// TwinCAT 3 PLC project Application
// ProgramVersion: 3.1.4022.2
// libraries:
//   Tc2_MC2, * (Beckhoff Automation GmbH)
//   Tc2_Standard, * (Beckhoff Automation GmbH)
//   Tc2_System, * (Beckhoff Automation GmbH)
//   Tc3_HBI_MC2, * (BeckHoff)
//   Tc3_Module, * (Beckhoff Automation GmbH)
// project tree:
//   / PlcTask.TcTTO
//   POUs/ MAIN.TcPOU, ST_Axis.TcDUT
// real-time tasks:
//   TASK PlcTask: cycle T#10ms, priority 20, ADS port 350
// motion (NC):
//   TASK NC-Task 1 SAF: cycle T#2ms, priority 4, ADS port 501
//   TASK NC-Task 1 SVB: cycle T#10ms, priority 8, ADS port 511
//   AXIS Axis 1 (id 1)
//     OtherSettings: AllowMotionCmdToSlave=true
//     encoder EncType=1
//     drive DrvType=5
//       Analog: ScaleFactorActTorque=0.1
//     controller CtrType=1
//       CtrPara: PriorControlFactor=1
//         Observer: BandWidth=20
//   AXIS Axis 2 (id 2)
//     OtherSettings: AllowMotionCmdToSlave=true
//     encoder EncType=1
//     drive DrvType=5
//       Analog: ScaleFactorActTorque=0.1
//     controller CtrType=1
//       CtrPara: PriorControlFactor=1
//         Observer: BandWidth=20
//   AXIS Axis 3 (id 3)
//     OtherSettings: AllowMotionCmdToSlave=true
//     encoder EncType=1
//     drive DrvType=5
//       Analog: ScaleFactorActTorque=0.1
//     controller CtrType=1
//       CtrPara: PriorControlFactor=1
//         Observer: BandWidth=20
// variable links:
//   Application/Application Instance <-> NC-Task 1 SAF/Axes/Axis 1
//     PlcTask Inputs/MAIN.fbAxis[0]._stAXIS_REF.NcToPlc <-> Outputs/ToPlc
//     PlcTask Outputs/MAIN.fbAxis[0]._stAXIS_REF.PlcToNc <-> Inputs/FromPlc
//   Application/Application Instance <-> NC-Task 1 SAF/Axes/Axis 2
//     PlcTask Inputs/MAIN.fbAxis[1]._stAXIS_REF.NcToPlc <-> Outputs/ToPlc
//     PlcTask Outputs/MAIN.fbAxis[1]._stAXIS_REF.PlcToNc <-> Inputs/FromPlc
//   Application/Application Instance <-> NC-Task 1 SAF/Axes/Axis 3
//     PlcTask Inputs/MAIN.fbAxis[2]._stAXIS_REF.NcToPlc <-> Outputs/ToPlc
//     PlcTask Outputs/MAIN.fbAxis[2]._stAXIS_REF.PlcToNc <-> Inputs/FromPlc

CONFIGURATION Application
    RESOURCE PLC ON TwinCAT3
        TASK PlcTask(INTERVAL := T#10ms, PRIORITY := 20);
        PROGRAM MAIN WITH PlcTask : MAIN;
    END_RESOURCE
END_CONFIGURATION

// ---- POUs/ST_Axis.TcDUT
TYPE ST_Axis :
STRUCT
	bEnable: BOOL;
	bEnable_Negative: BOOL;
	bEnable_Positive: BOOL;
	lrOverride: LREAL;
	bReset	: BOOL;
	bE_Stop: BOOL;
	bE_StopDelay: BOOL;
	bHome: BOOL;
	bCalibrationCam	: BOOL;
	lrHomePosition	: LREAL;
	bHalt	: BOOL;
	bStop	: BOOL;
	bAbsMove	: BOOL;
	lrAbsPosition	: LREAL;
	lrAbsVelocity	: LREAL;
	bRelMove	: BOOL;
	lrRelDistance	: LREAL;
	lrRelVelocity	: LREAL;
	bMoveVelo	: BOOL;
	lrVeloVelocity	: LREAL;
	bJogForward: BOOL;
	bJogBackwards: BOOL;
	lrJogVelocity	: LREAL;
	bSetDynamic		: BOOL;
	lrAcceleration	: LREAL;
	lrDecelaration	: LREAL;
	lrJerk			: LREAL;
	arr_nStatus	: ARRAY[1..10] OF UDINT;	

	//Vanessa added
	lrActPos : LREAL;
	lrActVelo : LREAL;
	bReady : BOOL;
	nVeloDirection : INT;
	nErrId : UDINT;
END_STRUCT
END_TYPE

// ---- POUs/MAIN.TcPOU
PROGRAM MAIN
VAR
	nAlive: INT;
	// Axis Instance
	fbAxis: ARRAY[0..2] OF Tc3_HBI_MC2.FB_MC2_Basic;
	
	bCalibrationCam : BOOL; //home sensor
	stAxis: ARRAY[0..2] OF ST_Axis;
	i: INT;
	
	//Input
	bInput1 : BOOL;
	bInput2 : BOOL;
	bInput3 : BOOL;
	bInput4 : BOOL;
	bInput5 : BOOL;
	bInput6 : BOOL;
	bInput7 : BOOL;
	bInput8 : BOOL;
	bInput9 : BOOL;
	bInput10 : BOOL;
	
	//Output
	bOutput1 : BOOL;
	bOutput2 : BOOL;
	bOutput3 : BOOL;
	bOutput4 : BOOL;
	bOutput5 : BOOL;
	bOutput6 : BOOL;
	bOutput7 : BOOL;
	bOutput8 : BOOL;
	bOutput9 : BOOL;
	bOutput10 : BOOL;
	
END_VAR

nAlive:= nAlive +1;

FOR i:= 0 TO 2 DO
	
//************************************
// Call methods
//************************************
stAxis[i].arr_nStatus[1]:= fbAxis[i].M_nMC_Power(bEnable:= stAxis[i].bEnable, bE_Stop:= stAxis[i].bE_Stop, 									// Enable
							bE_StopDelay:= stAxis[i].bE_StopDelay, bEnable_Positive:= stAxis[i].bEnable_Positive, 
							bEnable_Negative:= stAxis[i].bEnable_Negative);							
stAxis[i].arr_nStatus[2]:= fbAxis[i].M_nReset(bExecute:= stAxis[i].bReset);																// Reset
stAxis[i].arr_nStatus[3]:= fbAxis[i].M_nMC_Halt(bExecute:= stAxis[i].bHalt);																// Halt
stAxis[i].arr_nStatus[4]:= fbAxis[i].M_nMC_Stop(bExecute:= stAxis[i].bStop);																// Stop
stAxis[i].arr_nStatus[5]:= fbAxis[i].M_nMC_Home(bExecute:= stAxis[i].bHome, lrPosition:= stAxis[i].lrHomePosition, 							// Home
											bCalibrationCam:= stAxis[i].bCalibrationCam, eHomingMode:= MC_DefaultHoming);		
stAxis[i].arr_nStatus[6]:= fbAxis[i].M_nMC_MoveAbsolute(bExecute:= stAxis[i].bAbsMove, lrPosition:= stAxis[i].lrAbsPosition, 				// Absolute
													lrVelocity:= stAxis[i].lrAbsVelocity);									
stAxis[i].arr_nStatus[7]:= fbAxis[i].M_nMC_MoveRelative(bExecute:= stAxis[i].bRelMove, lrDistance:= stAxis[i].lrRelDistance, 				// Relative
													lrVelocity:= stAxis[i].lrRelVelocity);									
stAxis[i].arr_nStatus[8]:= fbAxis[i].M_nMC_Jog(bForward:= stAxis[i].bJogForward, bBackwards:= stAxis[i].bJogBackwards, 						// Jog 
											lrVelocity:= stAxis[i].lrJogVelocity);	
stAxis[i].arr_nStatus[9]:= fbAxis[i].M_nMC_Dynamic(bExecute:= stAxis[i].bSetDynamic, lrAcceleration:= stAxis[i].lrAcceleration, 			// Set dynamic
											lrDeceleration:= stAxis[i].lrDecelaration, lrJerk:= stAxis[i].lrJerk);		
stAxis[i].arr_nStatus[10]:= fbAxis[i].M_nMC_MoveVelocity(bExecute:= stAxis[i].bMoveVelo, lrVelocity:= stAxis[i].lrVeloVelocity, 			// Velocity
													eDirection:=  stAxis[i].nVeloDirection);								
													
													
// Home sensor
stAxis[i].bCalibrationCam:= bCalibrationCam;
stAxis[i].lrActPos := fbAxis[i]._stAXIS_REF.NcToPlc.ActPos;
stAxis[i].lrActVelo := fbAxis[i]._stAXIS_REF.NcToPlc.ActVelo;
stAxis[i].bReady := fbAxis[i].P_bReady;
stAxis[i].nErrId := fbAxis[i].P_nErrorID;

stAxis[i].bE_Stop := TRUE;
stAxis[i].bE_StopDelay := TRUE;
stAxis[i].lrJogVelocity := 100;

END_FOR

END_PROGRAM
